SUBAPPLICATION Uebung_088 (* Beispiel für E_F_TRIG *)
  (* Standard: 61499-2; Description: Copyright (c) 2023 Meisterschulen am Ostbahnhof This program and the accompanying materials are made available under the terms of the Eclipse Public License 2.0 which is available at https://www.eclipse.org/legal/epl-2.0/ SPDX-License-Identifier: EPL-2.0 *)
  (* Version 1.0, 2023-10-23, Franz Höpfinger, Meisterschulen am Ostbahnhof *)
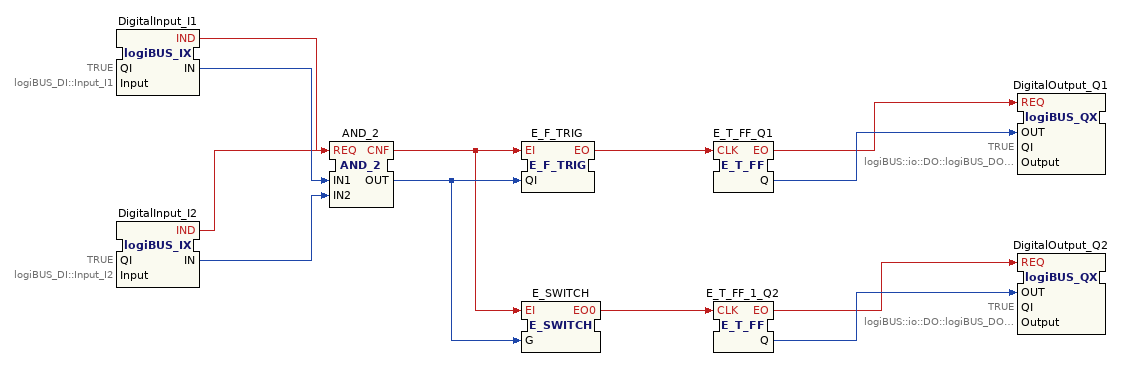
  (* F_TRIG schaltet nur wenn wirklich fallende Flanke *)
  (* E_SWITCH schaltet auch, wenn anderweitig ein Event kommt. *)
  FBS
    DigitalOutput_Q1 : logiBUS_QX(QI := TRUE, Output := logiBUS::io::DO::logiBUS_DO::Output_Q1);
    DigitalInput_I1 : logiBUS_IX(QI := TRUE, Input := logiBUS_DI::Input_I1);
    AND_2 : AND_2;
    DigitalInput_I2 : logiBUS_IX(QI := TRUE, Input := logiBUS_DI::Input_I2);
    E_F_TRIG : E_F_TRIG;
    E_T_FF_Q1 : E_T_FF;
    DigitalOutput_Q2 : logiBUS_QX(QI := TRUE, Output := logiBUS::io::DO::logiBUS_DO::Output_Q2);
    E_T_FF_1_Q2 : E_T_FF;
    E_SWITCH : E_SWITCH;
  END_FBS
  EVENT_CONNECTIONS
    DigitalInput_I2.IND TO AND_2.REQ;
    DigitalInput_I1.IND TO AND_2.REQ;
    AND_2.CNF TO E_F_TRIG.EI;
    E_F_TRIG.EO TO E_T_FF_Q1.CLK;
    E_T_FF_Q1.EO TO DigitalOutput_Q1.REQ;
    E_SWITCH.EO0 TO E_T_FF_1_Q2.CLK;
    AND_2.CNF TO E_SWITCH.EI;
    E_T_FF_1_Q2.EO TO DigitalOutput_Q2.REQ;
  END_CONNECTIONS
  DATA_CONNECTIONS
    DigitalInput_I1.IN TO AND_2.IN1;
    DigitalInput_I2.IN TO AND_2.IN2;
    AND_2.OUT TO E_F_TRIG.QI;
    E_T_FF_Q1.Q TO DigitalOutput_Q1.OUT;
    AND_2.OUT TO E_SWITCH.G;
    E_T_FF_1_Q2.Q TO DigitalOutput_Q2.OUT;
  END_CONNECTIONS
END_SUBAPPLICATION
